// TwinCAT 3 PLC project PLC_1
// ProgramVersion: 3.1.4024.0
// libraries:
//   SPT Base Types, * (Beckhoff Automation LLC)
//   SPT Components, * (Beckhoff Automation LLC)
//   Tc2_Standard, * (Beckhoff Automation GmbH)
//   Tc2_System, * (Beckhoff Automation GmbH)
//   Tc3_IPCDiag, * (Beckhoff Automation GmbH)
//   Tc3_JsonXml, * (Beckhoff Automation GmbH)
//   Tc3_Module, * (Beckhoff Automation GmbH)
// project tree:
//   / PlcTask.TcTTO
//   POUs/ MAIN.TcPOU
// real-time tasks:
//   TASK PlcTask: cycle T#10ms, priority 20, ADS port 350

CONFIGURATION PLC_1
    RESOURCE PLC ON TwinCAT3
        TASK PlcTask(INTERVAL := T#10ms, PRIORITY := 20);
        PROGRAM MAIN WITH PlcTask : MAIN;
    END_RESOURCE
END_CONFIGURATION

// ---- POUs/MAIN.TcPOU
PROGRAM MAIN
VAR
Sensor :FB_DigitalSensor;
Simulate :BOOL;
Activte :BOOL;
t1,t2 :TIME;
Traced :BOOL;
inData :BOOL;

END_VAR

// Konfiguracja czujnika
Sensor.SimulationMode := E_SensorSimulationMode.InputDriven;
Sensor.Name := 'My Sensor'; // Zamiana ' na właściwy apostrof '
Sensor.InSimulation := Simulate;
Sensor.SimulationInput := inData;

// Przypisanie wartości wyjść czujnika
Activte := Sensor.Active;
t1 := Sensor.TimeActive;
t2 := Sensor.TimeInactive;

// Cykl logiki czujnika
Sensor.CyclicLogic();

// Logika śledzenia
IF t1 >= T#5S THEN
    IF NOT Traced THEN
        Traced := TRUE;
        Sensor.Trace(Message := 'The sensor is on more than 5s'); // Zamiana ' na właściwy apostrof
    END_IF
ELSE
    Traced := FALSE;
END_IF

END_PROGRAM
